(* IEC 61131-3 sources: volt/packages/volt-lsp-iec/test-corpus/lenze-mid/Device/Plc Logic/Application/A55_VarLists/Safety, 6 files *)

(* ---- GVL_3.gvl ---- *)
{attribute 'qualified_only'}
VAR_GLOBAL
//SafetyStatus_01 :
ServiceButtonHasResetFunction : BOOL;
//SafetyStatus_01 :
FeedbackEstop : BOOL;
//SafetyStatus_01 :
FeedbackDoors : BOOL;
//SafetyStatus_01 :
FeedbackSTO : BOOL;
//SafetyStatus_01 :
ErrorInInputModule : BOOL;
//SafetyStatus_01 :
ErrorInOutputModule : BOOL;
//SafetyStatus_01 :
Emergency_button01 : BOOL;
//SafetyStatus_01 :
Emergency_button02 : BOOL;
//SafetyStatus_01 :
Emergency_button03 : BOOL;
//SafetyStatus_01 :
Emergency_button04 : BOOL;
//SafetyStatus_01 :
Emergency_button05 : BOOL;
//SafetyStatus_01 :
Emergency_button06 : BOOL;
//SafetyStatus_01 :
Emergency_input_upstream : BOOL;
//SafetyStatus_01 :
Emergency_input_downstream : BOOL;
//SafetyStatus_01 :
Emergency_output_upstream : BOOL;
//SafetyStatus_01 :
Emergency_output_downstream : BOOL;
END_VAR

(* ---- Safety_Status001.gvl ---- *)
{attribute 'qualified_only'}
VAR_GLOBAL
//SafetyStatus_00 :
EmergencyStopOK : BOOL;
//SafetyStatus_00 :
EmergencyStopDelayed : BOOL;
//SafetyStatus_00 :
DoorsOK : BOOL;
//SafetyStatus_00 :
DoorsDelayed : BOOL;
//SafetyStatus_00 :
ServiceMode : BOOL;
//SafetyStatus_00 :
SafetyAutoSpeed : BOOL;
//SafetyStatus_00 :
SafetyManSpeed : BOOL;
//SafetyStatus_00 :
STO_OK : BOOL;
//SafetyStatus_00 :
HoldDrive : BOOL;
//SafetyStatus_00 :
AllDoorsActuallyClosed : BOOL;
//SafetyStatus_00 :
CustomError2 : BOOL;
//SafetyStatus_00 :
CustomError3 : BOOL;
//SafetyStatus_00 :
Service_ButtonCD : BOOL;
//SafetyStatus_00 :
Service_ButtonAB : BOOL;
//SafetyStatus_00 :
EnableServiceMuting : BOOL;
//SafetyStatus_00 :
EnableMuting : BOOL;
END_VAR

(* ---- Safety_Status02.gvl ---- *)
{attribute 'qualified_only'}
VAR_GLOBAL
//SafetyStatus_02 :
Door_switch01 : BOOL;
//SafetyStatus_02 :
Door_switch02 : BOOL;
//SafetyStatus_02 :
Door_switch03 : BOOL;
//SafetyStatus_02 :
Door_switch04 : BOOL;
//SafetyStatus_02 :
Door_switch05 : BOOL;
//SafetyStatus_02 :
Door_switch06 : BOOL;
//SafetyStatus_02 :
Door_switch07 : BOOL;
//SafetyStatus_02 :
Door_switch08 : BOOL;
//SafetyStatus_02 :
Door_switch09 : BOOL;
//SafetyStatus_02 :
Door_switch10 : BOOL;
//SafetyStatus_02 :
Door_switch11 : BOOL;
//SafetyStatus_02 :
Door_switch12 : BOOL;
//SafetyStatus_02 :
Door_switch13 : BOOL;
//SafetyStatus_02 :
Door_switch14 : BOOL;
//SafetyStatus_02 :
Door_switch15 : BOOL;
//SafetyStatus_02 :
Door_switch16 : BOOL;
END_VAR

(* ---- Safety_Status03.gvl ---- *)
{attribute 'qualified_only'}
VAR_GLOBAL
//SafetyStatus_03 :
Door_switch17 : BOOL;
//SafetyStatus_03 :
Door_switch18 : BOOL;
//SafetyStatus_03 :
Door_switch19 : BOOL;
//SafetyStatus_03 :
Door_switch20 : BOOL;
//SafetyStatus_03 :
Door_switch21 : BOOL;
//SafetyStatus_03 :
Door_switch22 : BOOL;
//SafetyStatus_03 :
Door_switch23 : BOOL;
//SafetyStatus_03 :
Door_switch24 : BOOL;
//SafetyStatus_03 :
Door_switch25 : BOOL;
//SafetyStatus_03 :
Door_switch26 : BOOL;
//SafetyStatus_03 :
Door_switch27 : BOOL;
//SafetyStatus_03 :
Door_switch28 : BOOL;
//SafetyStatus_03 :
Door_switch29 : BOOL;
//SafetyStatus_03 :
Door_switch30 : BOOL;
//SafetyStatus_03 :
Door_switch31 : BOOL;
//SafetyStatus_03 :
Custom_ATF_Disabled : BOOL;
END_VAR

(* ---- SafetyControl_00.gvl ---- *)
{attribute 'qualified_only'}
VAR_GLOBAL
//SafetyControl_00 :
ResetSafetyGuard : BOOL;
//SafetyControl_00 :
ExternalReset : BOOL;
//SafetyControl_00 :
ExternalRequestResetSafetyModule : BOOL;
//SafetyControl_00 :
RequestManSpeed : BOOL;
//SafetyControl_00 :
RequestAutoSpeed : BOOL;
//SafetyControl_00 :
Muting_zone1 : BOOL;
//SafetyControl_00 :
Muting_zone2 : BOOL;
//SafetyControl_00 :
Muting_zone3 : BOOL;
//SafetyControl_00 :
PartialMuting1 : BOOL;
//SafetyControl_00 :
PartialMuting2 : BOOL;
//SafetyControl_00 :
PartialMuting3 : BOOL;
//SafetyControl_00 :
ResetCustomError1 : BOOL;
//SafetyControl_00 :
ResetCustomError2 : BOOL;
//SafetyControl_00 :
ResetCustomError3 : BOOL;
//SafetyControl_00 :
ForceOutputs : BOOL;
//SafetyControl_00 :
Set_Global_EstopError : BOOL;
END_VAR

(* ---- SafetyControl_01.gvl ---- *)
{attribute 'qualified_only'}
VAR_GLOBAL
//SafetyControl_01 :
Set_Local_EstopError : BOOL;
//SafetyControl_01 :
Set_Local_DoorsError : BOOL;
//SafetyControl_01 :
Set_Local_STOError : BOOL;
//SafetyControl_01 :
CTRL_Spare01 : BOOL;
//SafetyControl_01 :
CTRL_Spare02 : BOOL;
//SafetyControl_01 :
CTRL_Spare03 : BOOL;
//SafetyControl_01 :
CTRL_Spare04 : BOOL;
//SafetyControl_01 :
CTRL_Spare05 : BOOL;
//SafetyControl_01 :
CTRL_Spare06 : BOOL;
//SafetyControl_01 :
CTRL_Spare07 : BOOL;
//SafetyControl_01 :
CTRL_Spare08 : BOOL;
//SafetyControl_01 :
CTRL_Spare09 : BOOL;
//SafetyControl_01 :
CTRL_Spare10 : BOOL;
//SafetyControl_01 :
CTRL_Spare11 : BOOL;
//SafetyControl_01 :
CTRL_Spare12 : BOOL;
//SafetyControl_01 :
CTRL_Spare13 : BOOL;
END_VAR
